{attribute addProperty BoxType "EK1100-0000-0018"}
{attribute addProperty Id "Beckhoff_EL67xxEK1122Beckhoff_EL67xxEK1122_6F27A5BF162A_0001_EL6720_0000_0016EL6720_8C99EE5012816A_0002_EL6720_0000_0017EL6720_8C99EE5012816A_0003_EL6720_0000_0018EL6720_8C99EE5012816A_0004_EL6720_0000_0020EL6720_8C99EE5012816A_0005_EL6731_0000_0000EL6731_8C99EE5012816A_0006_EL6731_0001_0000EL6731_8C99EE5012816A_0007_EL6731_0000_0016EL6731_8C99EE5012816A_0008_EL6731_0000_0017EL6731_8C99EE5012816A_0009_EL6731_0000_0018EL6731_8C99EE5012816A_0010_EL6731_0000_0019EL6731_8C99EE5012816A_0011_EL6731_0000_0020EL6731_8C99EE5012816A_0012_EL6731_0000_0021EL6731_8C99EE5012816A_0013_EL6731_0000_0022EL6731_8C99EE5012816A_0014_EL6731_0000_0023EL6731_8C99EE5012816A_0015_EL6731_0000_0025EL6731_8C99EE5012816A_0016_EL6731_0100_0017EL6731_8C99EE5012816A_0017_EL6731_0100_0018EL6731_8C99EE5012816A_0018_EL6731_0100_0019EL6731_8C99EE5012816A_0019_EL6731_0100_0020EL6731_8C99EE5012816A_0020_EL6731_0100_0021EL6731_8C99EE5012816A_0021_EL6731_0100_0022EL6731_8C99EE5012816A_0022_EL6731_0100_0023EL6731_8C99EE5012816A_0023_EL6731_0100_0025EL6731_8C99EE5012816A_0024_EL6731_0010_0000EL6731_8C99EE5012816A_0025_EL6731_0010_0016EL6731_8C99EE5012816A_0026_EL6731_0010_0017EL6731_8C99EE5012816A_0027_EL6731_0010_0018EL6731_8C99EE5012816A_0028_EL6731_0010_0019EL6731_8C99EE5012816A_0029_EL6731_0010_0021EL6731_8C99EE5012816A_0030_EL6731_1003_0016EL6731_8C99EE5012816A_0031_EL6740_0010_0000EL6740_AABC74D88210.25A_0032_EL6740_0010_0001EL6740_AABC74D88210.25A_0033_EL6740_0010_0002EL6740_AABC74D88210.25A_0034_EL6751_0000_0000EL6751_8C99EE5012816A_0035_EL6751_0001_0000EL6751_8C99EE5012816A_0036_EL6751_0000_0016EL6751_8C99EE5012816A_0037_EL6751_0000_0017EL6751_8C99EE5012816A_0038_EL6751_0000_0018EL6751_8C99EE5012816A_0039_EL6751_0000_0019EL6751_8C99EE5012816A_0040_EL6751_0000_0021EL6751_8C99EE5012816A_0041_EL6751_0000_0022EL6751_8C99EE5012816A_0042_EL6751_0005_0022EL6751_8C99EE5012816A_0043_EL6751_0010_0000EL6751_8C99EE5012816A_0044_EL6751_0010_0017EL6751_8C99EE5012816A_0045_EL6751_0010_0018EL6751_8C99EE5012816A_0046_EL6751_0010_0019EL6751_8C99EE5012816A_0047_EL6751_0010_0021EL6751_8C99EE5012816A_0048_EL6752_0000_0000EL6752_8C99EE5012816A_0049_EL6752_0000_0016EL6752_8C99EE5012816A_0050_EL6752_0000_0017EL6752_8C99EE5012816A_0051_EL6752_0000_0018EL6752_8C99EE5012816A_0052_EL6752_0000_0019EL6752_8C99EE5012816A_0053_EL6752_0000_0020EL6752_8C99EE5012816A_0054_EL6752_0010_0000EL6752_8C99EE5012816A_0055_EL6752_0010_0016EL6752_8C99EE5012816A_0056_EL6752_0010_0017EL6752_8C99EE5012816A_0057_EL6752_0010_0018EL6752_8C99EE5012816A_0058_EL6752_0010_0020EL6752_8C99EE5012816A_0059_EL6784_0000_0016EL6784_B3418C2811414.25A_0060_EL6784_0000_0017EL6784_B3418C2811414.25A_0061_EL6784_0000_0018EL6784_B3418C2811414.25"}
{attribute addProperty CRC "770075973"}
{attribute addProperty SizeInBites "7644"}
{attribute addProperty SizeInBytes "955.5"}
TYPE Beckhoff_EL67xx_2DE66D45 EXTENDS EK1100_179A0949 :
STRUCT
	{attribute addProperty Name "Beckhoff_EL67xxEK1122"}
	Beckhoff_EL67xxEK1122 : Beckhoff_EL67xxEK1122_6F27A5BF;
	{attribute addProperty Name "A_0001_EL6720_0000_0016"}
	A_0001_EL6720_0000_0016 : EL6720_8C99EE50;
	{attribute addProperty Name "A_0002_EL6720_0000_0017"}
	A_0002_EL6720_0000_0017 : EL6720_8C99EE50;
	{attribute addProperty Name "A_0003_EL6720_0000_0018"}
	A_0003_EL6720_0000_0018 : EL6720_8C99EE50;
	{attribute addProperty Name "A_0004_EL6720_0000_0020"}
	A_0004_EL6720_0000_0020 : EL6720_8C99EE50;
	{attribute addProperty Name "A_0005_EL6731_0000_0000"}
	A_0005_EL6731_0000_0000 : EL6731_8C99EE50;
	{attribute addProperty Name "A_0006_EL6731_0001_0000"}
	A_0006_EL6731_0001_0000 : EL6731_8C99EE50;
	{attribute addProperty Name "A_0007_EL6731_0000_0016"}
	A_0007_EL6731_0000_0016 : EL6731_8C99EE50;
	{attribute addProperty Name "A_0008_EL6731_0000_0017"}
	A_0008_EL6731_0000_0017 : EL6731_8C99EE50;
	{attribute addProperty Name "A_0009_EL6731_0000_0018"}
	A_0009_EL6731_0000_0018 : EL6731_8C99EE50;
	{attribute addProperty Name "A_0010_EL6731_0000_0019"}
	A_0010_EL6731_0000_0019 : EL6731_8C99EE50;
	{attribute addProperty Name "A_0011_EL6731_0000_0020"}
	A_0011_EL6731_0000_0020 : EL6731_8C99EE50;
	{attribute addProperty Name "A_0012_EL6731_0000_0021"}
	A_0012_EL6731_0000_0021 : EL6731_8C99EE50;
	{attribute addProperty Name "A_0013_EL6731_0000_0022"}
	A_0013_EL6731_0000_0022 : EL6731_8C99EE50;
	{attribute addProperty Name "A_0014_EL6731_0000_0023"}
	A_0014_EL6731_0000_0023 : EL6731_8C99EE50;
	{attribute addProperty Name "A_0015_EL6731_0000_0025"}
	A_0015_EL6731_0000_0025 : EL6731_8C99EE50;
	{attribute addProperty Name "A_0016_EL6731_0100_0017"}
	A_0016_EL6731_0100_0017 : EL6731_8C99EE50;
	{attribute addProperty Name "A_0017_EL6731_0100_0018"}
	A_0017_EL6731_0100_0018 : EL6731_8C99EE50;
	{attribute addProperty Name "A_0018_EL6731_0100_0019"}
	A_0018_EL6731_0100_0019 : EL6731_8C99EE50;
	{attribute addProperty Name "A_0019_EL6731_0100_0020"}
	A_0019_EL6731_0100_0020 : EL6731_8C99EE50;
	{attribute addProperty Name "A_0020_EL6731_0100_0021"}
	A_0020_EL6731_0100_0021 : EL6731_8C99EE50;
	{attribute addProperty Name "A_0021_EL6731_0100_0022"}
	A_0021_EL6731_0100_0022 : EL6731_8C99EE50;
	{attribute addProperty Name "A_0022_EL6731_0100_0023"}
	A_0022_EL6731_0100_0023 : EL6731_8C99EE50;
	{attribute addProperty Name "A_0023_EL6731_0100_0025"}
	A_0023_EL6731_0100_0025 : EL6731_8C99EE50;
	{attribute addProperty Name "A_0024_EL6731_0010_0000"}
	A_0024_EL6731_0010_0000 : EL6731_8C99EE50;
	{attribute addProperty Name "A_0025_EL6731_0010_0016"}
	A_0025_EL6731_0010_0016 : EL6731_8C99EE50;
	{attribute addProperty Name "A_0026_EL6731_0010_0017"}
	A_0026_EL6731_0010_0017 : EL6731_8C99EE50;
	{attribute addProperty Name "A_0027_EL6731_0010_0018"}
	A_0027_EL6731_0010_0018 : EL6731_8C99EE50;
	{attribute addProperty Name "A_0028_EL6731_0010_0019"}
	A_0028_EL6731_0010_0019 : EL6731_8C99EE50;
	{attribute addProperty Name "A_0029_EL6731_0010_0021"}
	A_0029_EL6731_0010_0021 : EL6731_8C99EE50;
	{attribute addProperty Name "A_0030_EL6731_1003_0016"}
	A_0030_EL6731_1003_0016 : EL6731_8C99EE50;
	{attribute addProperty Name "A_0031_EL6740_0010_0000"}
	A_0031_EL6740_0010_0000 : EL6740_AABC74D8;
	{attribute addProperty Name "A_0032_EL6740_0010_0001"}
	A_0032_EL6740_0010_0001 : EL6740_AABC74D8;
	{attribute addProperty Name "A_0033_EL6740_0010_0002"}
	A_0033_EL6740_0010_0002 : EL6740_AABC74D8;
	{attribute addProperty Name "A_0034_EL6751_0000_0000"}
	A_0034_EL6751_0000_0000 : EL6751_8C99EE50;
	{attribute addProperty Name "A_0035_EL6751_0001_0000"}
	A_0035_EL6751_0001_0000 : EL6751_8C99EE50;
	{attribute addProperty Name "A_0036_EL6751_0000_0016"}
	A_0036_EL6751_0000_0016 : EL6751_8C99EE50;
	{attribute addProperty Name "A_0037_EL6751_0000_0017"}
	A_0037_EL6751_0000_0017 : EL6751_8C99EE50;
	{attribute addProperty Name "A_0038_EL6751_0000_0018"}
	A_0038_EL6751_0000_0018 : EL6751_8C99EE50;
	{attribute addProperty Name "A_0039_EL6751_0000_0019"}
	A_0039_EL6751_0000_0019 : EL6751_8C99EE50;
	{attribute addProperty Name "A_0040_EL6751_0000_0021"}
	A_0040_EL6751_0000_0021 : EL6751_8C99EE50;
	{attribute addProperty Name "A_0041_EL6751_0000_0022"}
	A_0041_EL6751_0000_0022 : EL6751_8C99EE50;
	{attribute addProperty Name "A_0042_EL6751_0005_0022"}
	A_0042_EL6751_0005_0022 : EL6751_8C99EE50;
	{attribute addProperty Name "A_0043_EL6751_0010_0000"}
	A_0043_EL6751_0010_0000 : EL6751_8C99EE50;
	{attribute addProperty Name "A_0044_EL6751_0010_0017"}
	A_0044_EL6751_0010_0017 : EL6751_8C99EE50;
	{attribute addProperty Name "A_0045_EL6751_0010_0018"}
	A_0045_EL6751_0010_0018 : EL6751_8C99EE50;
	{attribute addProperty Name "A_0046_EL6751_0010_0019"}
	A_0046_EL6751_0010_0019 : EL6751_8C99EE50;
	{attribute addProperty Name "A_0047_EL6751_0010_0021"}
	A_0047_EL6751_0010_0021 : EL6751_8C99EE50;
	{attribute addProperty Name "A_0048_EL6752_0000_0000"}
	A_0048_EL6752_0000_0000 : EL6752_8C99EE50;
	{attribute addProperty Name "A_0049_EL6752_0000_0016"}
	A_0049_EL6752_0000_0016 : EL6752_8C99EE50;
	{attribute addProperty Name "A_0050_EL6752_0000_0017"}
	A_0050_EL6752_0000_0017 : EL6752_8C99EE50;
	{attribute addProperty Name "A_0051_EL6752_0000_0018"}
	A_0051_EL6752_0000_0018 : EL6752_8C99EE50;
	{attribute addProperty Name "A_0052_EL6752_0000_0019"}
	A_0052_EL6752_0000_0019 : EL6752_8C99EE50;
	{attribute addProperty Name "A_0053_EL6752_0000_0020"}
	A_0053_EL6752_0000_0020 : EL6752_8C99EE50;
	{attribute addProperty Name "A_0054_EL6752_0010_0000"}
	A_0054_EL6752_0010_0000 : EL6752_8C99EE50;
	{attribute addProperty Name "A_0055_EL6752_0010_0016"}
	A_0055_EL6752_0010_0016 : EL6752_8C99EE50;
	{attribute addProperty Name "A_0056_EL6752_0010_0017"}
	A_0056_EL6752_0010_0017 : EL6752_8C99EE50;
	{attribute addProperty Name "A_0057_EL6752_0010_0018"}
	A_0057_EL6752_0010_0018 : EL6752_8C99EE50;
	{attribute addProperty Name "A_0058_EL6752_0010_0020"}
	A_0058_EL6752_0010_0020 : EL6752_8C99EE50;
	{attribute addProperty Name "A_0059_EL6784_0000_0016"}
	A_0059_EL6784_0000_0016 : EL6784_B3418C28;
	{attribute addProperty Name "A_0060_EL6784_0000_0017"}
	A_0060_EL6784_0000_0017 : EL6784_B3418C28;
	{attribute addProperty Name "A_0061_EL6784_0000_0018"}
	A_0061_EL6784_0000_0018 : EL6784_B3418C28;
END_STRUCT
END_TYPE

(* stored: Version 1.2.0.0, ProductVersion 3.1.4024.9
   DUT Beckhoff_EL67xx_2DE66D45: Id {61c136ea-7332-4271-898d-14870357153b} *)
